Staubli VAL3: SavePreset.pgx

public program SavePreset(bool& x_bRes (dimensions=1))
  local num l_nNum
  local num l_nY
  local string l_sFileName
  local string l_sSBuff
begin


  //参数初始化
  x_bRes=false
  l_sFileName="Disk://Txt/Preset.txt"


  //关闭所有文件
  call FileDir:CloseAllFile()


  //文件是否可以打开
  nFileID=$fileOpen(l_sFileName,"w")
  if nFileID<0 or nFileID>9
    return
  endIf

  l_sSBuff="PRESET=StaubliPreset"
  if $fileSet(nFileID,l_sSBuff,1)!=1
    return
  endIf
  for l_nNum=1 to 50
    //最小是0，最大是100
    for l_nY=0 to 4
      nPreset[l_nNum,l_nY]=min(100,max(0,nPreset[l_nNum,l_nY]))
    endFor

    //直接输出
    l_sSBuff=toString("",nPreset[l_nNum,0])+","+toString("",nPreset[l_nNum,1])+","+toString("",nPreset[l_nNum,2])+","
    l_sSBuff=l_sSBuff+toString("",nPreset[l_nNum,3])+","+toString("",nPreset[l_nNum,4])
    if $fileSet(nFileID,l_sSBuff,1)!=1
      return
    endIf
  endFor
  call FileDir:CloseAllFile()

  x_bRes=true

end
